// Mitsubishi GX Works2 project: R&D&A 2.5   PLC: FX3G

// global labels: Global1
VAR_GLOBAL
  X_7 AT X007 : BOOL;
  Y_7 AT Y007 : BOOL;
  emergency_button AT X003 : BOOL;
  M_STOP AT M13 : BOOL;
  M_1 AT M1 : BOOL;
  no_inventory AT M3 : BOOL;
  M_blink_3sec AT M5 : BOOL;
  begginingBiscuit AT D1109 : REAL;
  begginingChoco AT D1117 : REAL;
  begginingKatzefet AT D1107 : REAL;
  currentBiscuit AT D1103 : REAL;
  currentChco AT D1105 : REAL;
  currentKatzefet AT D1101 : REAL;
  X_1 AT X001 : BOOL;
  M_0 AT M0 : BOOL;
END_VAR
VAR_GLOBAL CONSTANT
  minKatzefet : REAL := 300;
  minBiscuit : REAL := 6;
  minChco : REAL := 120;
END_VAR
VAR_GLOBAL
  M_2 AT M2 : BOOL;
  M_4 AT M4 : BOOL;
  X_11 AT X011 : BOOL;
END_VAR
VAR_GLOBAL CONSTANT
  c_300 : REAL := 300;
  minminBiscuit : REAL := 6;
  minminKatzefet : REAL := 300;
END_VAR
VAR_GLOBAL
  M_9 AT M9 : BOOL;
  M_10 AT M10 : BOOL;
  TS_1 AT TS1 : BOOL;
  TC_1 AT TC1 : BOOL;
END_VAR
VAR_GLOBAL CONSTANT
  CON_20 : INT;
END_VAR
VAR_GLOBAL
  M_200 AT M200 : BOOL;
  TC_2 AT TC2 : BOOL;
  TS_2 AT TS2 : BOOL;
  M_300 AT M300 : BOOL;
  TS_5 AT TS5 : BOOL;
  M_19 AT M19 : BOOL;
  TC_5 AT TC5 : BOOL;
  Y_5 AT Y005 : BOOL;
END_VAR
VAR_GLOBAL CONSTANT
  CON_30 : INT := 30;
END_VAR
VAR_GLOBAL
  TC_3 AT TC3 : BOOL;
END_VAR
VAR_GLOBAL CONSTANT
  CON_40 : INT := 40;
  CON_CON_4040 : INT := 40;
END_VAR
VAR_GLOBAL
  TS_3 AT TS3 : BOOL;
  Y_0 AT Y000 : BOOL;
  Y_1 AT Y001 : BOOL;
  M_17 AT M17 : BOOL;
END_VAR
VAR_GLOBAL CONSTANT
  CON_4 : INT := 40;
END_VAR
VAR_GLOBAL
  M_150 AT M150 : BOOL;
  TC_7 AT TC7 : BOOL;
  TS_7 AT TS7 : BOOL;
  X_6 AT X006 : BOOL;
  analogInput1 AT D8280 : INT;
  M_18 AT M18 : BOOL;
END_VAR
VAR_GLOBAL CONSTANT
  minDoubleChoco : REAL := 240;
END_VAR
VAR_GLOBAL
  M_14 AT M14 : BOOL;
  M_24 AT M24 : BOOL;
END_VAR
VAR_GLOBAL CONSTANT
  CONSTANT_395 : INT := 395;
  con5 : INT := 5;
END_VAR
VAR_GLOBAL
  M_26 AT M26 : BOOL;
  TC_24 AT TC24 : BOOL;
  TS_24 AT TS24 : BOOL;
END_VAR
VAR_GLOBAL CONSTANT
  CON_50 : INT := 50;
END_VAR
VAR_GLOBAL
  Y_3 AT Y003 : BOOL;
  x_0 AT X000 : BOOL;
  cc_1 AT CC1 : BOOL;
END_VAR
VAR_GLOBAL CONSTANT
  CO_5 : INT := 5;
END_VAR
VAR_GLOBAL
  cs_1 AT CS1 : BOOL;
  y_2 AT Y002 : BOOL;
  cc3 AT CC3 : BOOL;
END_VAR
VAR_GLOBAL CONSTANT
  CO_6 : INT := 6;
END_VAR
VAR_GLOBAL
  cs_3 AT CS3 : BOOL;
  x_10 AT X010 : BOOL;
END_VAR
VAR_GLOBAL CONSTANT
  sdfsdgfd : REAL := 1000;
END_VAR
VAR_GLOBAL
  M_30 AT M30 : BOOL;
  analogOUTPUT AT D8282 : INT;
  x_4 AT X004 : BOOL;
  beggingKatzefet AT D1107 : REAL;
END_VAR
VAR_GLOBAL CONSTANT
  fhjut : REAL := 1000;
  startWith1000 : REAL := 1000;
END_VAR
VAR_GLOBAL
  endOfRound AT M32 : BOOL;
  analogInputNirmul1 AT D7000 : INT;
  CN_1 AT CN1 : INT;
  CN_3 AT CN3 : INT;
END_VAR
VAR_GLOBAL CONSTANT
  CO_1 : INT := 1;
END_VAR
VAR_GLOBAL
  TC_9 AT TC9 : BOOL;
  M_32 AT M32 : BOOL;
  forResetDay AT M32 : BOOL;
END_VAR
VAR_GLOBAL CONSTANT
  CON_5 : INT := 5;
END_VAR
VAR_GLOBAL
  Y_4 AT Y004 : BOOL;
  m_240m240 AT M240 : BOOL;
END_VAR
VAR_GLOBAL CONSTANT
  CON_39 : INT := 39;
  CON_195 : INT := 195;
  startWithCHOCO : REAL := 300;
END_VAR
VAR_GLOBAL
  TC_11 AT TC11 : BOOL;
  TS_11 AT TS11 : BOOL;
  TS_9 AT TS9 : BOOL;
END_VAR

// task Task_01 (event TRUE, interval 0, priority 31): POU_01

PROGRAM POU_01
(* structured ladder/FBD written out as ST: instructions are called as NAME(EN, inputs, outputs); _pN, _eN, _tN stand for wires *)
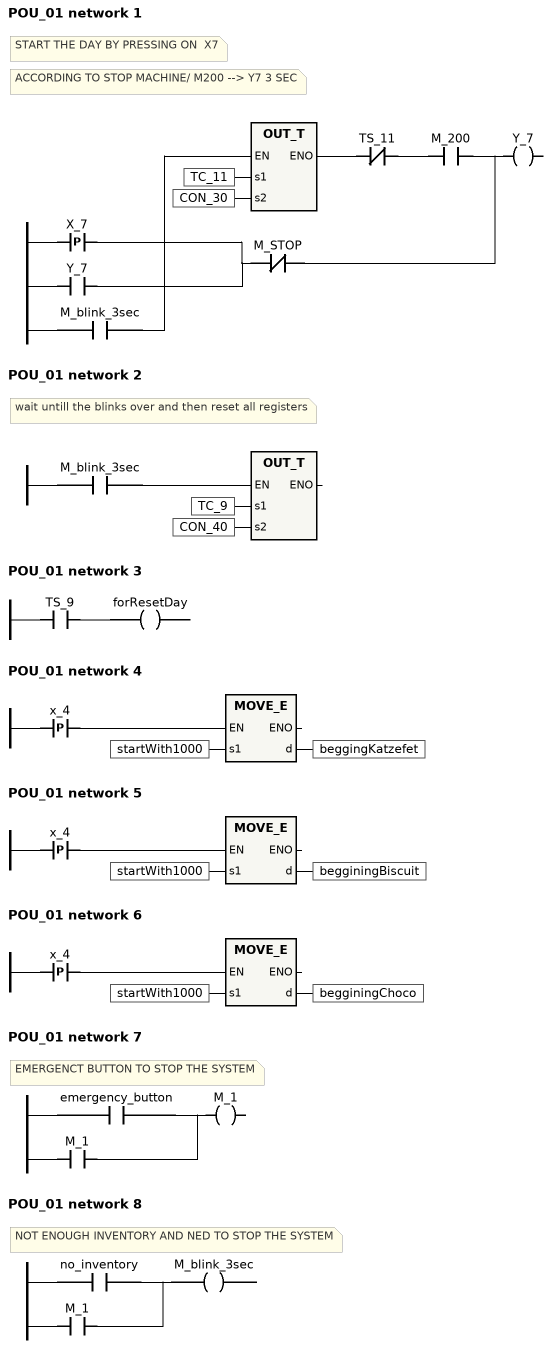
(* network 1 *)
(* START THE DAY BY PRESSING ON  X7 *)
(* ACCORDING TO STOP MACHINE/ M200 --> Y7 3 SEC *)
_e1 := OUT_T(M_blink_3sec, TC_11, CON_30);
Y_7 := ((LDP(TRUE, X_7) OR Y_7) AND NOT M_STOP) OR (_e1 AND NOT TS_11 AND M_200);
(* network 2 *)
(* wait untill the blinks over and then reset all registers *)
OUT_T(M_blink_3sec, TC_9, CON_40);
(* network 3 *)
forResetDay := TS_9;
(* network 4 *)
MOVE_E(LDP(TRUE, x_4), startWith1000, beggingKatzefet);
(* network 5 *)
MOVE_E(LDP(TRUE, x_4), startWith1000, begginingBiscuit);
(* network 6 *)
MOVE_E(LDP(TRUE, x_4), startWith1000, begginingChoco);
(* network 7 *)
(* EMERGENCT BUTTON TO STOP THE SYSTEM *)
M_1 := emergency_button OR M_1;
(* network 8 *)
(* NOT ENOUGH INVENTORY AND NED TO STOP THE SYSTEM *)
M_blink_3sec := no_inventory OR M_1;
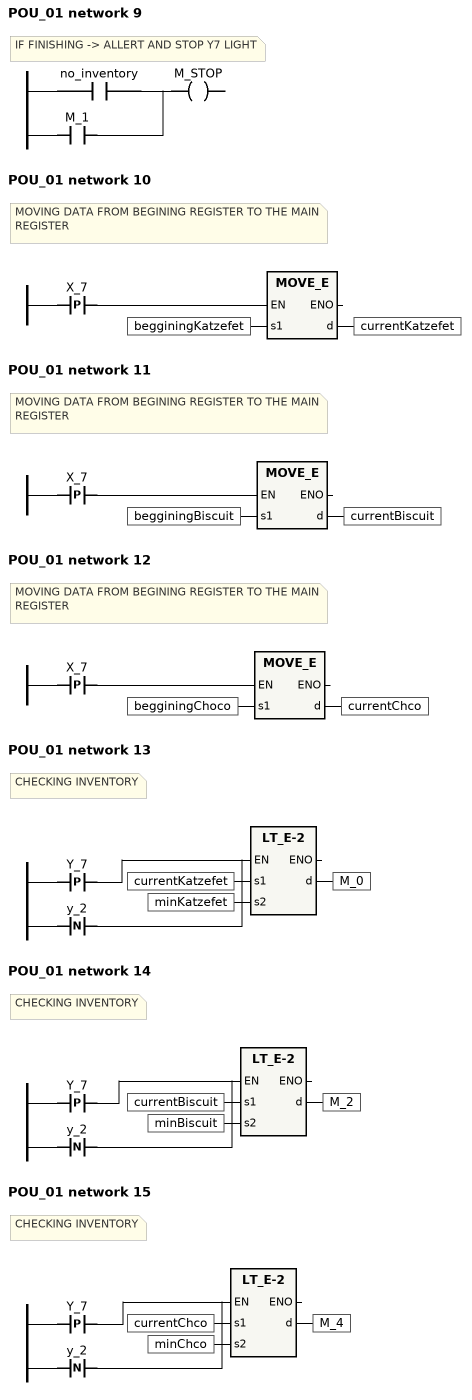
(* network 9 *)
(* IF FINISHING -> ALLERT AND STOP Y7 LIGHT *)
M_STOP := no_inventory OR M_1;
(* network 10 *)
(* MOVING DATA FROM BEGINING REGISTER TO THE MAIN REGISTER *)
MOVE_E(LDP(TRUE, X_7), begginingKatzefet, currentKatzefet);
(* network 11 *)
(* MOVING DATA FROM BEGINING REGISTER TO THE MAIN REGISTER *)
MOVE_E(LDP(TRUE, X_7), begginingBiscuit, currentBiscuit);
(* network 12 *)
(* MOVING DATA FROM BEGINING REGISTER TO THE MAIN REGISTER *)
MOVE_E(LDP(TRUE, X_7), begginingChoco, currentChco);
(* network 13 *)
(* CHECKING INVENTORY *)
LT_E(LDP(TRUE, Y_7) OR LDF(TRUE, y_2), currentKatzefet, minKatzefet, M_0);
(* network 14 *)
(* CHECKING INVENTORY *)
LT_E(LDP(TRUE, Y_7) OR LDF(TRUE, y_2), currentBiscuit, minBiscuit, M_2);
(* network 15 *)
(* CHECKING INVENTORY *)
LT_E(LDP(TRUE, Y_7) OR LDF(TRUE, y_2), currentChco, minChco, M_4);
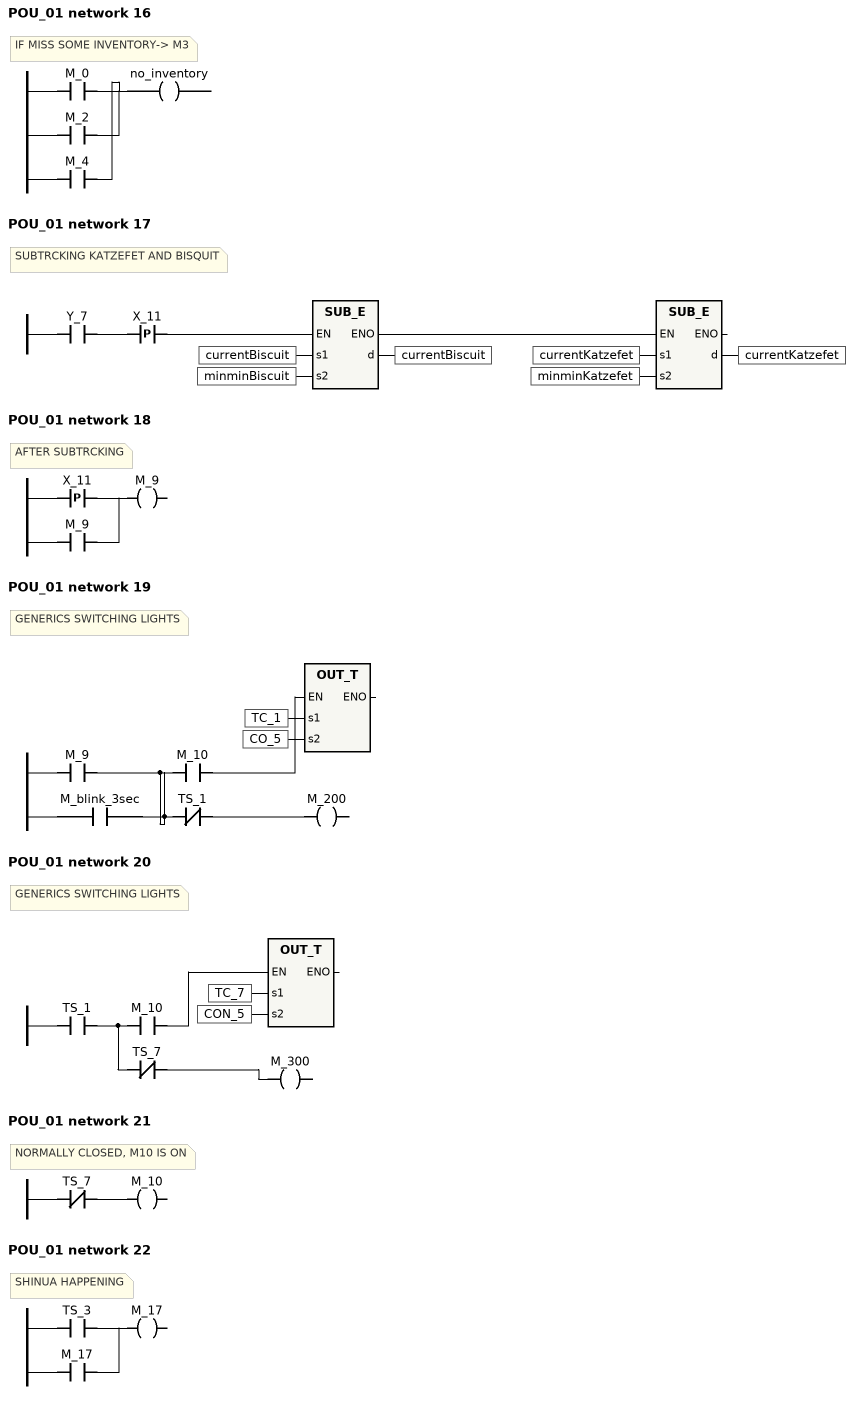
(* network 16 *)
(* IF MISS SOME INVENTORY-> M3 *)
no_inventory := M_0 OR M_2 OR M_4;
(* network 17 *)
(* SUBTRCKING KATZEFET AND BISQUIT *)
_e1 := SUB_E(Y_7 AND LDP(TRUE, X_11), currentBiscuit, minminBiscuit, currentBiscuit);
SUB_E(_e1, currentKatzefet, minminKatzefet, currentKatzefet);
(* network 18 *)
(* AFTER SUBTRCKING *)
M_9 := LDP(TRUE, X_11) OR M_9;
(* network 19 *)
(* GENERICS SWITCHING LIGHTS *)
_p1 := M_9 OR M_blink_3sec;
OUT_T(_p1 AND M_10, TC_1, CO_5);
M_200 := _p1 AND NOT TS_1;
(* network 20 *)
(* GENERICS SWITCHING LIGHTS *)
OUT_T(TS_1 AND M_10, TC_7, CON_5);
M_300 := TS_1 AND NOT TS_7;
(* network 21 *)
(* NORMALLY CLOSED, M10 IS ON *)
M_10 := NOT TS_7;
(* network 22 *)
(* SHINUA HAPPENING *)
M_17 := TS_3 OR M_17;
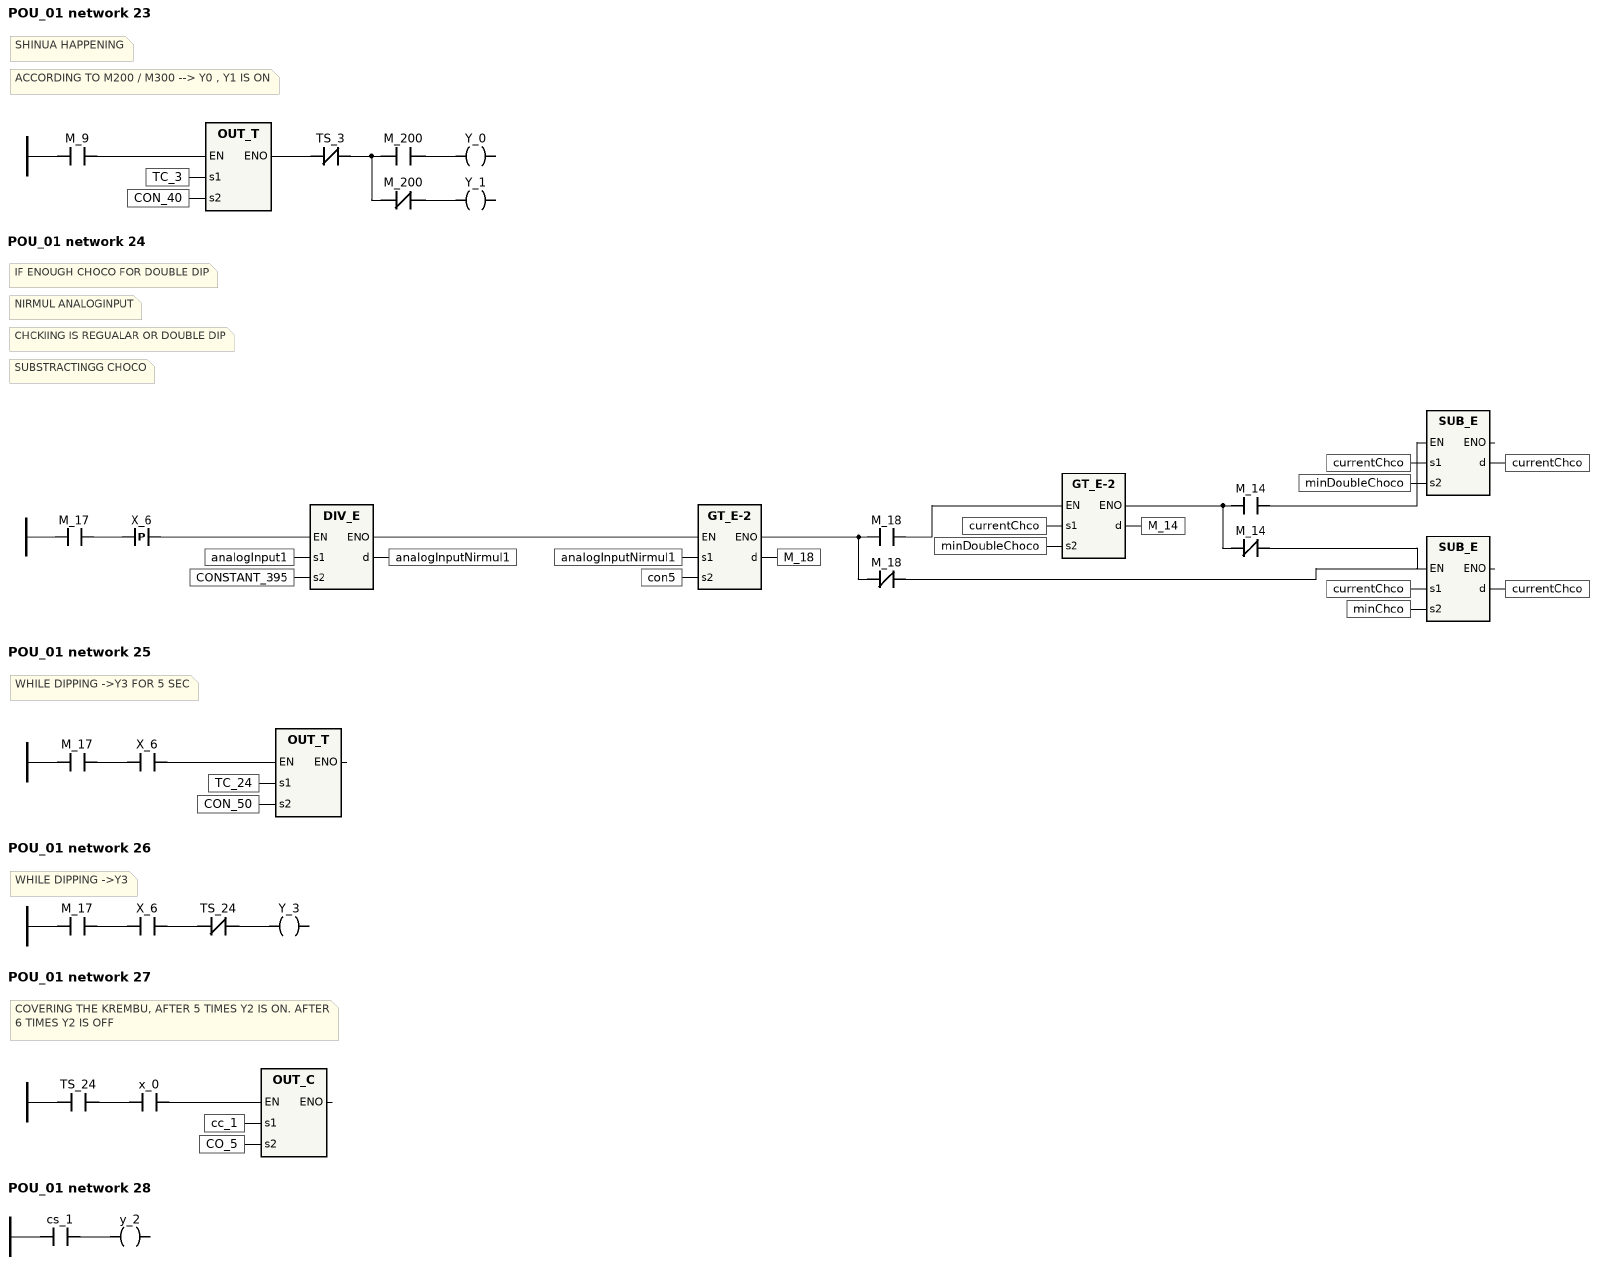
(* network 23 *)
(* SHINUA HAPPENING *)
(* ACCORDING TO M200 / M300 --> Y0 , Y1 IS ON *)
_e1 := OUT_T(M_9, TC_3, CON_40);
_p2 := _e1 AND NOT TS_3;
Y_0 := _p2 AND M_200;
Y_1 := _p2 AND NOT M_200;
(* network 24 *)
(* IF ENOUGH CHOCO FOR DOUBLE DIP *)
(* NIRMUL ANALOGINPUT *)
(* CHCKIING IS REGUALAR OR DOUBLE DIP *)
(* SUBSTRACTINGG CHOCO *)
_e1 := DIV_E(M_17 AND LDP(TRUE, X_6), analogInput1, CONSTANT_395, analogInputNirmul1);
_e2 := GT_E(_e1, analogInputNirmul1, con5, M_18);
_e3 := GT_E(_e2 AND M_18, currentChco, minDoubleChoco, M_14);
SUB_E(_e3 AND M_14, currentChco, minDoubleChoco, currentChco);
SUB_E((_e3 AND NOT M_14) OR (_e2 AND NOT M_18), currentChco, minChco, currentChco);
(* network 25 *)
(* WHILE DIPPING ->Y3 FOR 5 SEC *)
OUT_T(M_17 AND X_6, TC_24, CON_50);
(* network 26 *)
(* WHILE DIPPING ->Y3 *)
Y_3 := M_17 AND X_6 AND NOT TS_24;
(* network 27 *)
(* COVERING THE KREMBU, AFTER 5 TIMES Y2 IS ON. AFTER 6 TIMES Y2 IS OFF *)
OUT_C(TS_24 AND x_0, cc_1, CO_5);
(* network 28 *)
y_2 := cs_1;
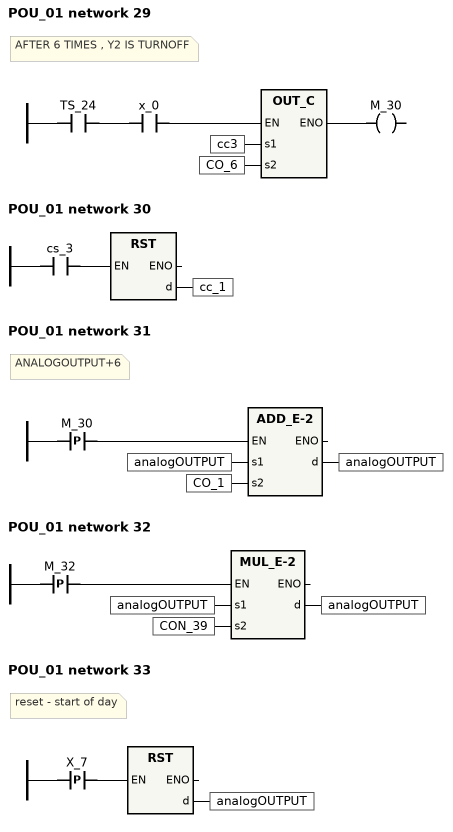
(* network 29 *)
(* AFTER 6 TIMES , Y2 IS TURNOFF *)
_e1 := OUT_C(TS_24 AND x_0, cc3, CO_6);
M_30 := _e1;
(* network 30 *)
RST(cs_3, cc_1);
(* network 31 *)
(* ANALOGOUTPUT+6 *)
ADD_E(LDP(TRUE, M_30), analogOUTPUT, CO_1, analogOUTPUT);
(* network 32 *)
MUL_E(LDP(TRUE, M_32), analogOUTPUT, CON_39, analogOUTPUT);
(* network 33 *)
(* reset - start of day *)
RST(LDP(TRUE, X_7), analogOUTPUT);
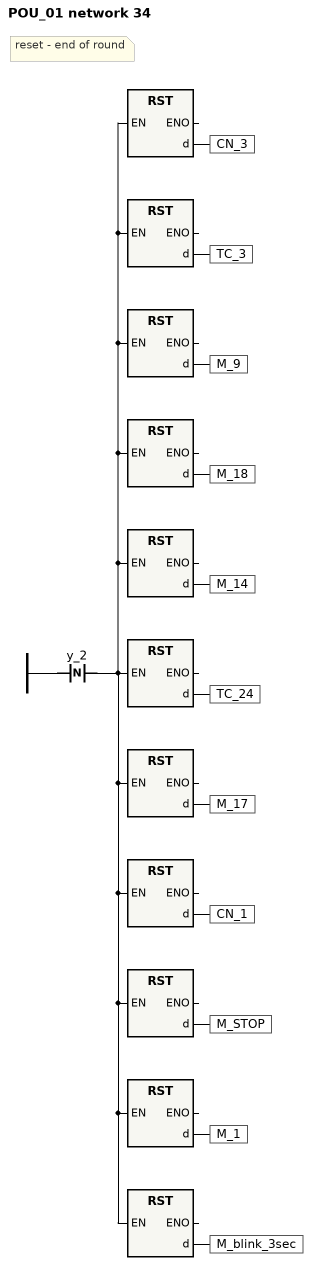
(* network 34 *)
(* reset - end of round *)
_p1 := LDF(TRUE, y_2);
RST(_p1, CN_3);
RST(_p1, TC_3);
RST(_p1, M_9);
RST(_p1, M_18);
RST(_p1, M_14);
RST(_p1, TC_24);
RST(_p1, M_17);
RST(_p1, CN_1);
RST(_p1, M_STOP);
RST(_p1, M_1);
RST(_p1, M_blink_3sec);
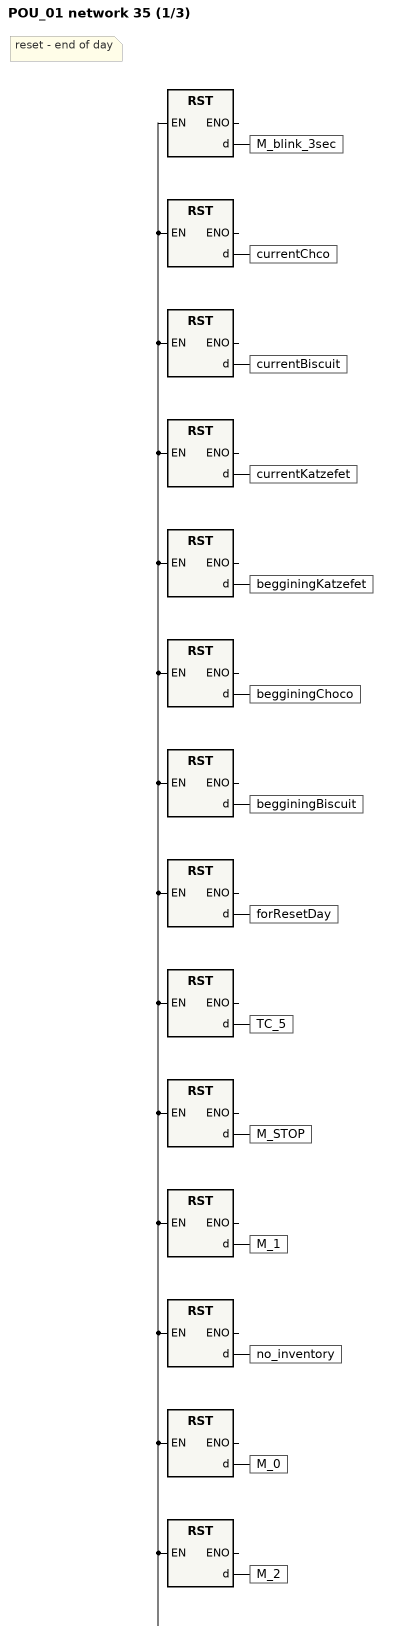
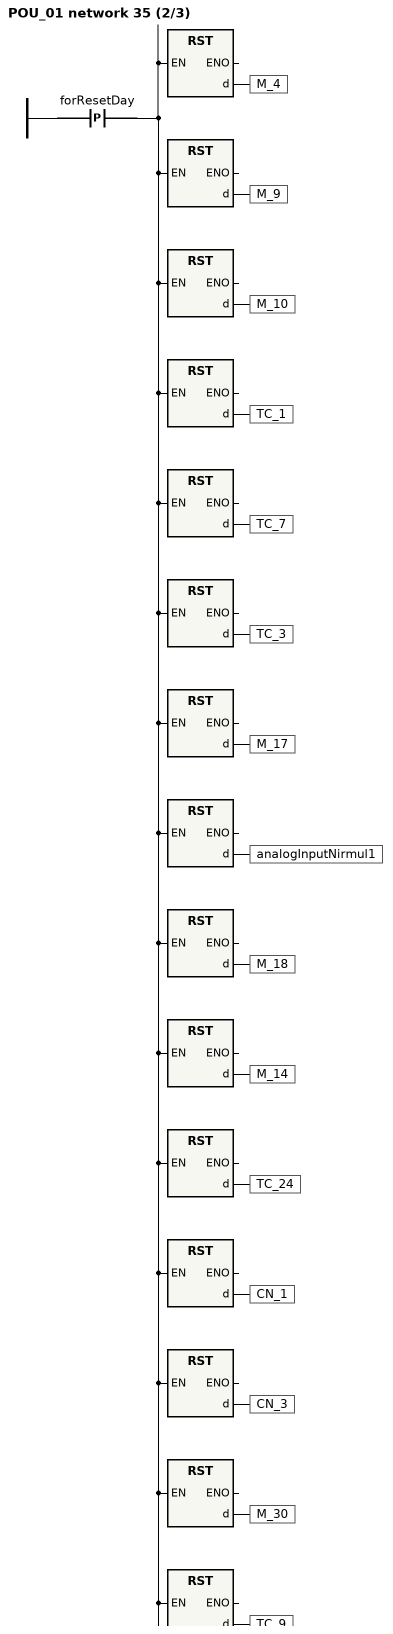
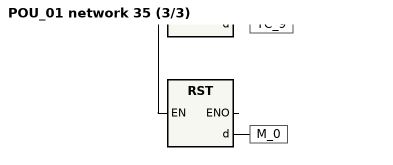
(* network 35 *)
(* reset - end of day *)
_p1 := LDP(TRUE, forResetDay);
RST(_p1, M_blink_3sec);
RST(_p1, currentChco);
RST(_p1, currentBiscuit);
RST(_p1, currentKatzefet);
RST(_p1, begginingKatzefet);
RST(_p1, begginingChoco);
RST(_p1, begginingBiscuit);
RST(_p1, forResetDay);
RST(_p1, TC_5);
RST(_p1, M_STOP);
RST(_p1, M_1);
RST(_p1, no_inventory);
RST(_p1, M_0);
RST(_p1, M_2);
RST(_p1, M_4);
RST(_p1, M_9);
RST(_p1, M_10);
RST(_p1, TC_1);
RST(_p1, TC_7);
RST(_p1, TC_3);
RST(_p1, M_17);
RST(_p1, analogInputNirmul1);
RST(_p1, M_18);
RST(_p1, M_14);
RST(_p1, TC_24);
RST(_p1, CN_1);
RST(_p1, CN_3);
RST(_p1, M_30);
RST(_p1, TC_9);
RST(_p1, M_0);
END_PROGRAM
